{attribute addProperty BoxType "AT2050-0500-0022"}
{attribute addProperty Id "A_0091_AT2020_5250_0017_AT2020_5250AT2020_C5E5984862678.25"}
{attribute addProperty CRC "1241416301"}
{attribute addProperty SizeInBites "626"}
{attribute addProperty SizeInBytes "78.25"}
TYPE A_0053_AT2050_0500_0022_49FE826D EXTENDS AT2050_BA5A9548 :
STRUCT
	{attribute addProperty Name "A_0091_AT2020_5250_0017_AT2020_5250"}
	A_0091_AT2020_5250_0017_AT2020_5250 : AT2020_C5E59848;
END_STRUCT
END_TYPE

(* stored: Version 1.2.0.0, ProductVersion 3.1.4024.9
   DUT A_0053_AT2050_0500_0022_49FE826D: Id {8b89d723-e12a-4677-b660-9aa3a5cf0dac} *)
